{attribute 'GeneratedUsingTerminal: EK1122-0000-0018'}
{attribute addProperty BoxType "EK1122-0000-0018"}
{attribute addProperty Id "Beckhoff_EL37xxsub_EK1100EK1100_1FC0878B2"}
{attribute addProperty CRC "562016005"}
{attribute addProperty Size "2"}
TYPE Beckhoff_EL37xxEK1122_217FAF05 EXTENDS EK1122_1FC0878B :
STRUCT
	{attribute addProperty Name "Beckhoff_EL37xxsub_EK1100"}
	{attribute addProperty PreviousPort "Beckhoff EL37xxEK1122 : D"}
	Beckhoff_EL37xxsub_EK1100 : EK1100_1FC0878B;
END_STRUCT
END_TYPE

(* stored: Version 1.2.0.0, ProductVersion 3.1.4024.9
   DUT Beckhoff_EL37xxEK1122_217FAF05: Id {1df9cb7b-b914-4fdb-a757-77a5e929880e} *)
